(* CODESYS project PiPlate_MOTOR.library
   Company: Lennart
   DefaultNamespace: PiPlate_MOTOR
   Title: PiPlate_MOTOR
   Placeholder: PlaceholderTemplate
   Author: Lennart Albertsen
   Description: Library containing device support of PiPlate DAQC Digital
   Version: 1.2.0.0

Project tree, tasks and I/O mapping:
  libraries: IoDrvGPIO, * (3S - Smart Software Solutions GmbH); Raspberry Pi Peripherals, * (3S - Smart Software Solutions GmbH); IoStandard, * (System)
  global variables GCL_PiPlate_MOTOR
  00000000-0000-0000-0000-000000000000|D:\CoDeSys\LibrariesV3\trunk\Intern\CAA\CAA Template\3.4.0.0 draft\Placeholder.xml
  00000000-0000-0000-0000-000000000000|D:\CoDeSys\LibrariesV3\trunk\Intern\CAA\CAA Template\3.2.0.3 draft\Prefix.pdf
  00000000-0000-0000-0000-000000000000|D:\CoDeSys\LibrariesV3\trunk\Intern\CAA\CAA Template\3.5.2.0 draft\Placeholder.xml
  function block PiPlate_MOTOR [ST]: Initialize, BeforeWriteOutputs, AfterReadInputs, read8, write8
  function block STEPPER [ST]: Initialize
  data type MOTOR_dt
  data type STEPPER_dt
  function block DC_Motor [ST]
*)

// MOTOR_dt
TYPE MOTOR_dt :
STRUCT
	Start:BOOL;
	SpeedSp:LREAL;
	SpeedAct:LREAL;
END_STRUCT
END_TYPE

// STEPPER_dt
TYPE STEPPER_dt :
STRUCT
	Pos:LREAL;
	ActPos:LREAL;
	Conf:BYTE;
END_STRUCT
END_TYPE

// GCL_PiPlate_MOTOR
VAR_GLOBAL CONSTANT
	//OUTPUT_PORT: USINT := 16#0D;
	//INPUT_PORT: USINT := 16#19;
	//IOCON: USINT := 0;
	//GPIOA: USINT := 16#14;
	//GPIOB: USINT := 16#13;
	//GPPUB: USINT := 16#0D;
	//IODIRA: USINT := 16#00;
	//IODIRB: USINT := 16#01;
DELAY_SETTLE_NS : UDINT := 40000; // 40us
DELAY_SETTLE_NSX : UDINT := 400000; // 400us
END_VAR

// PiPlate_MOTOR
FUNCTION_BLOCK PiPlate_MOTOR EXTENDS spi
VAR_INPUT
	//DO1:BOOL; //Digital Output 1
	//DO2:BOOL; //Digital Output 2
	//DO3:BOOL; //Digital Output 3
	//DO4:BOOL; //Digital Output 4
	//DO5:BOOL; //Digital Output 5
	//DO6:BOOL; //Digital Output 6
	//DO7:BOOL; //Digital Output 7
	//AO1:UINT; //Analog Output 1 Range: 0..1023
	//AO2:UINT; //Analog Output 2 Range: 0..1023
	Stepper1Conf:ARRAY[0..3] OF BYTE; (*Direction,resolution,rate,acceleration*)
	Stepper1Move:UINT; (*Steps*)
	Stepper1Jog:BOOL; (*Jog*)
	Stepper2Conf:ARRAY[0..3] OF BYTE; (*Direction,resolution,rate,acceleration*)
	Stepper2Move:UINT; (*Steps*)
	Stepper2Jog:BOOL; (*Jog*)

END_VAR
VAR_OUTPUT
	//DI1:BOOL; //Digital Input 1
	//DI2:BOOL; //Digital Input 2
	//DI3:BOOL; //Digital Input 3
	//DI4:BOOL; //Digital Input 4
	//DI5:BOOL; //Digital Input 5
	//DI6:BOOL; //Digital Input 6
	//DI7:BOOL; //Digital Input 7
	//DI8:BOOL; //Digital Input 8
	//AI1:UINT; //Analog Input 1 Range: 0..1023
	//AI2:UINT; //Analog Input 2 Range: 0..1023
	//AI3:UINT; //Analog Input 3 Range: 0..1023
	//AI4:UINT; //Analog Input 4 Range: 0..1023
	//AI5:UINT; //Analog Input 5 Range: 0..1023
	//AI6:UINT; //Analog Input 6 Range: 0..1023
	//AI7:UINT; //Analog Input 7 Range: 0..1023
	//AI8:UINT; //Analog Input 8 Range: 0..1023
	MoveStepper1Done:BOOL;
	MoveStepper2Done:BOOL;
	OPR:BOOL; //Operational
END_VAR
VAR
	_byHardwareAddress: BYTE;
	BoardBaseAddress:BYTE :=16;
	BoardType:ARRAY [0..20] OF BYTE :=[0,0,0,0,80,105,45,80,108,97,116,101,32,77,79,84,79,82,0,0,0]; (*Pi-Plate MOTOR*)
	digitalOut:BYTE;
	digitalIn:BYTE;
	byInDO:BYTE;
	vState:INT;
	IOStatusOK:BOOL := TRUE;
	vRecArray:ARRAY [0..20] OF BYTE;
	PWMArray:ARRAY  [0..2] OF BYTE;
	vConfigTest:BOOL;
	vMotorMoveStart:BOOL;
	Steps:WORD;
	Increment:INT;
	Resolution:BYTE (0..3);
	Direction:BOOL;
	Rate:WORD (1..2000) :=100;
	Param1:BYTE;
	Param2:BYTE;
	Steps1:BYTE;
	Steps2:BYTE;
	Motor0State:BYTE;
	Motor1State:BYTE;
END_VAR
VAR_IN_OUT
	Stepper1Connect:STEPPER_dt;
	Stepper2Connect:STEPPER_dt;
	Motor1Connect:MOTOR_dt;
	Motor2Connect:MOTOR_dt;
	Motor3Connect:MOTOR_dt;
	Motor4Connect:MOTOR_dt;
END_VAR
VAR_TEMP
	i, k: INT;
END_VAR

SUPER^();

CASE _iState OF
0:	IF SUPER^.init() THEN
		read8(_byHardwareAddress,00,0,0,1); //Check Control Board Address
		IF vRecArray[4] = _byHardwareAddress + BoardBaseAddress THEN
			read8(_byHardwareAddress,01,0,0,1); //Check Control Board Type
			IF vRecArray[4] = BoardType[4] AND vRecArray[5] = BoardType[5] AND vRecArray[6] = BoardType[6] AND vRecArray[7] = BoardType[7] AND vRecArray[8] = BoardType[8] AND vRecArray[9] = BoardType[9] AND vRecArray[10] = BoardType[10] AND vRecArray[11] = BoardType[11] AND vRecArray[12] = BoardType[12] AND vRecArray[13] = BoardType[13] AND vRecArray[14] = BoardType[14] AND vRecArray[15] = BoardType[15] AND vRecArray[16] = BoardType[16] AND vRecArray[17] = BoardType[17] THEN
				_iState := 1;
			END_IF
		END_IF;
	END_IF	
1: 	_iState := 10;

10: //Board Present an OK
	IF _pConnector^.dwFlags = 242 OR NOT IOStatusOK THEN
	_iState:=1000;
	END_IF
	//write8(_byHardwareAddress,98,0,0,0); //Toggle LED
1000: _iState:=0;
END_CASE
OPR := Operational AND _iState = 10;

METHOD Initialize : UDINT
VAR_INPUT
	wModuleType : UINT;
	dwInstance : UDINT;
	pConnector : POINTER TO IoConfigConnector;
END_VAR
VAR
	pParam: POINTER TO IoConfigParameter;		
	udiResult: UDINT;
END_VAR
SUPER^.Initialize(wModuleType, dwInstance, pConnector);

pParam := ConfigGetParameter(_pConnector, 1);
IF pParam <> 0 THEN
	_byHardwareAddress := IoStandard.ConfigGetParameterValueByte(pParam, ADR(udiResult));
END_IF
END_METHOD

METHOD BeforeWriteOutputs : INT
VAR
	i: INT;

END_VAR
SUPER^.BeforeWriteOutputs();

IF _iState = 10 THEN

CASE vState OF
	0:	Param1 := WORD_TO_BYTE(Rate / 256) + SHL(Resolution,4);
		Param1.6 := Direction;
		Param2 := WORD_TO_BYTE(Rate);
		IF vConfigTest THEN
		//Write Configurstion To Stepper
			write8(_byHardwareAddress,16,Param1,Param2,0);
			//write8(_byHardwareAddress,17,Param1,Param2,0);
			vConfigTest := FALSE;
			vState := 1;
		END_IF;
		
		
	1:	Steps1 := WORD_TO_BYTE((Steps /256));
		Steps2 := WORD_TO_BYTE(Steps);
		IF vMotorMoveStart THEN
			write8(_byHardwareAddress,18,Steps1,Steps2,0);
			//write8(_byHardwareAddress,19,Steps1,Steps2,0);
			vMotorMoveStart := FALSE;
			vState := 2;
		END_IF;
		
	2:	read8(_byHardwareAddress,6,0,0,1);
		Motor0State := vRecArray[4];
		read8(_byHardwareAddress,6,0,0,1);
		Motor1State := vRecArray[4];
		vState := 3;
	
END_CASE


	
(*
Param1 := WORD_TO_BYTE(Rate / 256) + SHL(Resolution,4);
Param1.6 := Direction;
Param2 := WORD_TO_BYTE(Rate);
IF vConfigTest THEN
//Write Configurstion To Stepper
write8(_byHardwareAddress,16,Param1,Param2,0);
vConfigTest := FALSE;
END_IF;
Steps1 := WORD_TO_BYTE((Steps /256));
Steps2 := WORD_TO_BYTE(Steps);
IF vMotorMoveStart THEN
	write8(_byHardwareAddress,18,Steps1,Steps2,0);
	vMotorMoveStart := FALSE;
END_IF;
	*)
(*
		CASE vState OF
	
			0: 	read8(_byHardwareAddress,37,0,0,1); // Get Digital Inputs
				digitalIn := NOT vRecArray[4]; // DI inputs status
				DI1 := digitalIn.0;
				DI2 := digitalIn.1;
				DI3 := digitalIn.2;
				DI4 := digitalIn.3;
				DI5 := digitalIn.4;
				DI6 := digitalIn.5;
				DI7 := digitalIn.6;
				DI8 := digitalIn.7;
				vState := 1;	
		
			1: 	digitalOut.0 := DO1;
				digitalOut.1 := DO2;	
				digitalOut.2 := DO3;
				digitalOut.3 := DO4;
				digitalOut.4 := DO5;
				digitalOut.5 := DO6;
				digitalOut.6 := DO7;
				write8(_byHardwareAddress,19,digitalout,0,0); //Write Digital Outputs
				vState := 2;
				
			2: 	read8(_byHardwareAddress,20,0,0,1); // Get Digital Output status
				byInDO := vRecArray[4]; //DO's status feedback
				IOStatusOK := byInDO = digitalout;
				vState := 3;
		
			3: 	read8(_byHardwareAddress,49,1,0,16); // Get Analog Inputs
				AI1 := 256*vRecArray[4]+vRecArray[5]; //AI1 calc 0..1024
				AI2 := 256*vRecArray[6]+vRecArray[7]; //AI2 calc 0..1024
				AI3 := 256*vRecArray[8]+vRecArray[9]; //AI3 calc 0..1024
				AI4 := 256*vRecArray[10]+vRecArray[11]; //AI4 calc 0..1024
				AI5 := 256*vRecArray[12]+vRecArray[13]; //AI5 calc 0..1024
				AI6 := 256*vRecArray[14]+vRecArray[15]; //AI6 calc 0..1024
				AI7 := 256*vRecArray[16]+vRecArray[17]; //AI7 calc 0..1024
				AI8 := 256*vRecArray[18]+vRecArray[19]; //AI8 calc 0..1024
				vState := 4;
		
			4:	PWMArray[0] := UINT_TO_BYTE(AO1 /256);
				PWMArray[1] := UINT_TO_BYTE(AO1);
				write8(_byHardwareAddress,64,PWMArray[0],PWMArray[1],0); //write Analog Out1/PWM
				vState := 5;
		
			5:	PWMArray[0] := UINT_TO_BYTE(AO2 /256);
				PWMArray[1] := UINT_TO_BYTE(AO2);
				write8(_byHardwareAddress,65,PWMArray[0],PWMArray[1],0); //write Analog Out1/PWM
				vState := 0;
		END_CASE*)
END_IF
END_METHOD

METHOD AfterReadInputs : INT
VAR
END_VAR
SUPER^.AfterReadInputs();
END_METHOD

// This method is used to read the data byte of one port using the following protocol:
// Byte0: hardware address + 8
// Byte1: Command
// Byte2: Parameter1
// Byte3: Parameter2
// Bytes to return are written to vRecArray
METHOD read8 : BYTE
VAR_INPUT
	byHardwareAddress: BYTE (0..7); (* hardware address *)
	CMD : BYTE;
	PARAM1 : BYTE;
	PARAM2 : BYTE;
	Bytes2return:BYTE;
END_VAR
VAR
	abyTxBuffer: ARRAY [0..3] OF BYTE;
	abyRxBuffer: ARRAY [0..20] OF BYTE;
	i:INT;
END_VAR
abyTxBuffer[0] := byHardwareAddress +16; //SPI_WRITE_CMD;
abyTxBuffer[1] := CMD;
abyTxBuffer[2] := PARAM1;
abyTxBuffer[3] := PARAM2;


IF bytes2return > 0 THEN
	IF transferExt(pabyTxBuffer:=ADR(abyTxBuffer) , pabyRxBuffer:=ADR(abyRxBuffer) , udiSpeedHz:=25000 , udiLen:=20 , uiDelayus:=5) THEN
		vRecArray := abyRxBuffer;
	ELSE
	_iState := 1000;	
	END_IF 
END_IF
END_METHOD

// This method is used to write a data byte into a port using the following protocol:
// Byte0: hardware address + 8
// Byte1: Command
// Byte2: Parameter1
// Byte3: Parameter2
// Bytes to return (not used here)
METHOD write8 : BOOL
VAR_INPUT
	byHardwareAddress: BYTE (0..7); (* hardware address *)
	CMD : BYTE;
	PARAM1 : BYTE;
	PARAM2 : BYTE;
	Bytes2return:BYTE;
	
END_VAR
VAR_OUTPUT
	
END_VAR
VAR
	abyTxBuffer: ARRAY [0..3] OF BYTE;
	abyRxTBuffer: ARRAY [0..20] OF BYTE;
	i:INT;
	y:DWORD;
END_VAR
abyTxBuffer[0] := byHardwareAddress +16; //SPI_WRITE_CMD;
abyTxBuffer[1] := CMD;
abyTxBuffer[2] := PARAM1;
abyTxBuffer[3] := PARAM2;
	
write8 := transferExt(pabyTxBuffer:=ADR(abyTxBuffer) , pabyRxBuffer:=ADR(abyRxTBuffer) , udiSpeedHz:=500000 , udiLen:=4 , uiDelayus:=1);

IF NOT write8 THEN
   _iState := 1000;
END_IF
END_METHOD

END_FUNCTION_BLOCK

// STEPPER
FUNCTION_BLOCK STEPPER EXTENDS spi
VAR_INPUT
	Stepper_Conf:ARRAY[0..3] OF BYTE; (*Direction,resolution,rate,acceleration*)
	Stepper_Move:UINT; (*Steps*)
	Stepper_Jog:BOOL; (*Jog*)
END_VAR
VAR_OUTPUT
	MoveStepper_Done:BOOL;
END_VAR
VAR_IN_OUT
	StepperConnect:STEPPER_dt;
END_VAR
VAR
	Param1:BYTE;
	Param2:BYTE;
	NextParam1:BYTE;
	NextParam2:BYTE;
	Increment:INT;
	Resolution:BYTE (0..3);
	Direction:BOOL;
	Rate:WORD (1..2000);
	Acceleration:INT (0..10) :=1;
	_byHardwareAddress: BYTE;
	x: LREAL;
	pParam: Pointer to IoConfigParameter;	
	pPiPlate_STEPPER: POINTER TO STEPPER;
	usiAxisIndex: USINT;
	lrMinPos, lrMaxPos: LREAL;
	lrInitPos: LREAL;
END_VAR
VAR_TEMP
	i, k: INT;
END_VAR

SUPER^();
_iState:= 10;

	
//RATE0-7

Param1 := WORD_TO_BYTE(Rate / 256) + SHL(Resolution,4);
Param1.6 := Direction;
Param2 := WORD_TO_BYTE(Rate);
//Write Configurstion To Stepper
Increment := REAL_TO_INT((1024*Rate/(Acceleration*2000) +0.5));
NextParam1 := INT_TO_BYTE(Increment /256);
NextParam1.7 :=TRUE;
NextParam2 := INT_TO_BYTE(Increment);// & 255;
//RATE8-10
//Paramx := SHL(vResolution,4) + SHR(vRATE,8);
//Paramx := Param2 + SHL(Param1,8);
//BYTE Param2


NextParam1.0;
NextParam1.1;
NextParam1.2;
NextParam1.3;
NextParam1.4;
NextParam1.5;
NextParam1.6;
NextParam1.7;
Param2.0; //RATE0 
Param2.1; //RATE1
Param2.2; //RATE2
Param2.3; //RATE3
Param2.4; //RATE4
Param2.5; //RATE5
Param2.6; //RATE6
Param2.7; //RATE7 0..255
//BYTE Param1
Param1.0;  //RATE8
Param1.1;  //RATE9
Param1.2; //RATE10 0..127
Param1.3; //NA
Param1.4; //RES2
Param1.5; //RES1 0..3
Param1.6; //DIR  0..1
Param1.7; //0

METHOD Initialize : UDINT
VAR_INPUT
	wModuleType : UINT;
	dwInstance : UDINT;
	pConnector : POINTER TO IoConfigConnector;
END_VAR
VAR
	pParam: POINTER TO IoConfigParameter;		
	udiResult: UDINT;
END_VAR
SUPER^.Initialize(wModuleType, dwInstance, pConnector);

pParam := ConfigGetParameter(_pConnector, 1);
IF pParam <> 0 THEN
	_byHardwareAddress := IoStandard.ConfigGetParameterValueByte(pParam, ADR(udiResult));
END_IF
END_METHOD

END_FUNCTION_BLOCK

// DC_Motor
FUNCTION_BLOCK DC_Motor
VAR_INPUT
	setSpeed:LREAL;
END_VAR
VAR_IN_OUT
	MotorConnect:MOTOR_dt;
END_VAR
VAR
END_VAR

END_FUNCTION_BLOCK
